FUNCTION_BLOCK WP_Sensor_Single (* Basic Function Block Type *)
  (* Standard: 61499-2 *)
  (* Version 0.0, 2/7/2012, XPMUser, nxtControl GmbH, Template *)
  PACKAGE Main;
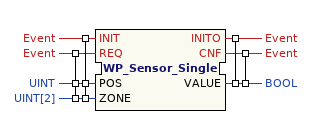
  EVENT_INPUT
    INIT WITH POS, ZONE; (* Initialization Request *)
    REQ WITH POS, ZONE; (* Normal Execution Request *)
  END_EVENT
  EVENT_OUTPUT
    INITO WITH VALUE; (* Initialization Confirm *)
    CNF WITH VALUE; (* Execution Confirmation *)
  END_EVENT
  VAR_INPUT
    POS : UINT; (* Input event qualifier *)
    ZONE : ARRAY [0..1] OF UINT;
  END_VAR
  VAR_OUTPUT
    VALUE : BOOL; (* Output event qualifier *)
  END_VAR
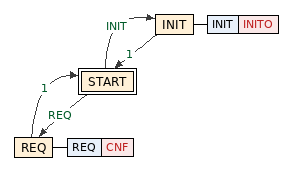
  EC_STATES
    START; (* Initial State *)
    INIT : INIT -> INITO; (* Initialization *)
    REQ : REQ -> CNF; (* Normal execution *)
  END_STATES
  EC_TRANSITIONS
    START TO INIT := INIT;
    INIT TO START := 1;
    START TO REQ := REQ;
    REQ TO START := 1;
  END_TRANSITIONS
  ALGORITHM INIT IN ST: (* Initialization algorithm *)
VALUE:=FALSE;
  END_ALGORITHM
  ALGORITHM REQ IN ST: (* Normally executed algorithm *)
IF POS >= ZONE[0] AND POS <= ZONE[1] THEN
    VALUE := TRUE;
ELSE
    VALUE := FALSE;
END_IF;
  END_ALGORITHM
END_FUNCTION_BLOCK
